// TIA Portal project "babu_counterBasics" (V15)

(* hardware
DEVICE "S7-1200 station_1"  S7-1200 Station
   slot 0: "Rack_0"  S7-1200 Rack  Rack  V1.0
   slot 1: "PLC_1"  CPU 1212C DC/DC/DC  6ES7 212-1AE40-0XB0  V4.2
*)

// ===== PLC "PLC_1"  CPU 1212C DC/DC/DC =====

VAR_GLOBAL   // PLC tag table "Default tag table"
   "sensor" AT %M0.0 : Bool;
   "reset" AT %M0.1 : Bool;
   "Tag_3" AT %MW0 : Int;
   "indicator light" AT %Q0.0 : Bool;
   "load" AT %M0.2 : Bool;
   "START PULSE 2" AT %M2.0 : Bool;
   "PULSE OUTPUT 2" AT %M2.1 : Bool;
   "START MEMORY" AT %M2.2 : Bool;
   "START MEMORY 2" AT %M2.3 : Bool;
   "TIMER MEMORY" AT %M2.4 : Bool;
   "COUNTER UP OUTPUT" AT %Q0.1 : Bool;
   "RESET CU" AT %M2.5 : Bool;
   "COUNTER DOWN OUTPUT" AT %Q0.2 : Bool;
   "LOAD DATA COUNTER DOWN" AT %M2.6 : Bool;
   "INITIALIZE" AT %M2.7 : Bool;
   "COUNTER UP DOWN OUTPUT" AT %M3.0 : Bool;
   "COUNTER DOWN RESET 5" AT %M3.1 : Bool;
   "COUNTER DOWN LOAD 5" AT %M3.2 : Bool;
   "COUNTER UP DOWN RESET" AT %M3.3 : Bool;
   "COUNTER DOWN 5" AT %M3.4 : Bool;
   "COUNTER DOWN OUTPUT 5" AT %M3.5 : Bool;
   "COUNTER DOWN SET 5" AT %M3.6 : Bool;
   "START 6" AT %M3.7 : Bool;
   "UP DOWN LONG PULSE" AT %M4.0 : Bool;
   "UP DOWN LONG PULSE MEM" AT %M4.1 : Bool;
   "COUNT UP" AT %M4.2 : Bool;
   "COUNT DOWN" AT %M4.3 : Bool;
   "COUNT DOWN TEMP" AT %M4.4 : Bool;
   "COUNTER UP OUTPUT 5" AT %M4.5 : Bool;
END_VAR

// folder: System blocks/Program resources

DATA_BLOCK "IEC_Counter_0_DB"   // DB1
{ S7_Optimized_Access := 'TRUE' }
AUTHOR : Simatic
FAMILY : IEC
NAME : CNTR
VERSION : 1.0
// stored: InstanceOfName IEC_COUNTER
"IEC_COUNTER"
BEGIN
END_DATA_BLOCK

DATA_BLOCK "IEC_Timer_0_DB_2"   // DB2
{ S7_Optimized_Access := 'TRUE' }
AUTHOR : Simatic
FAMILY : IEC
NAME : IEC_TMR
VERSION : 1.0
// stored: InstanceOfName IEC_TIMER
"IEC_TIMER"
BEGIN
END_DATA_BLOCK

DATA_BLOCK "IEC_Timer_0_DB"   // DB3
{ S7_Optimized_Access := 'TRUE' }
AUTHOR : Simatic
FAMILY : IEC
NAME : IEC_TMR
VERSION : 1.0
// stored: InstanceOfName IEC_TIMER
"IEC_TIMER"
BEGIN
END_DATA_BLOCK

DATA_BLOCK "IEC_Timer_0_DB_1"   // DB4
{ S7_Optimized_Access := 'TRUE' }
AUTHOR : Simatic
FAMILY : IEC
NAME : IEC_TMR
VERSION : 1.0
// stored: InstanceOfName IEC_TIMER
"IEC_TIMER"
BEGIN
END_DATA_BLOCK

DATA_BLOCK "IEC_Counter_0_DB_1"   // DB5
{ S7_Optimized_Access := 'TRUE' }
AUTHOR : Simatic
FAMILY : IEC
NAME : CNTR
VERSION : 1.0
// stored: InstanceOfName IEC_COUNTER
"IEC_COUNTER"
BEGIN
END_DATA_BLOCK

DATA_BLOCK "IEC_Timer_0_DB_3"   // DB6
{ S7_Optimized_Access := 'TRUE' }
AUTHOR : Simatic
FAMILY : IEC
NAME : IEC_TMR
VERSION : 1.0
// stored: InstanceOfName IEC_TIMER
"IEC_TIMER"
BEGIN
END_DATA_BLOCK

DATA_BLOCK "IEC_Counter_0_DB_2"   // DB7
{ S7_Optimized_Access := 'TRUE' }
AUTHOR : Simatic
FAMILY : IEC
NAME : CNTR
VERSION : 1.0
// stored: InstanceOfName IEC_COUNTER
"IEC_COUNTER"
BEGIN
END_DATA_BLOCK

DATA_BLOCK "IEC_Timer_0_DB_4"   // DB8
{ S7_Optimized_Access := 'TRUE' }
AUTHOR : Simatic
FAMILY : IEC
NAME : IEC_TMR
VERSION : 1.0
// stored: InstanceOfName IEC_TIMER
"IEC_TIMER"
BEGIN
END_DATA_BLOCK

DATA_BLOCK "IEC_Timer_0_DB_5"   // DB9
{ S7_Optimized_Access := 'TRUE' }
AUTHOR : Simatic
FAMILY : IEC
NAME : IEC_TMR
VERSION : 1.0
// stored: InstanceOfName IEC_TIMER
"IEC_TIMER"
BEGIN
END_DATA_BLOCK

DATA_BLOCK "IEC_Counter_0_DB_3"   // DB10
{ S7_Optimized_Access := 'TRUE' }
AUTHOR : Simatic
FAMILY : IEC
NAME : CNTR
VERSION : 1.0
// stored: InstanceOfName IEC_COUNTER
"IEC_COUNTER"
BEGIN
END_DATA_BLOCK

DATA_BLOCK "IEC_Timer_0_DB_6"   // DB11
{ S7_Optimized_Access := 'TRUE' }
AUTHOR : Simatic
FAMILY : IEC
NAME : IEC_TMR
VERSION : 1.0
// stored: InstanceOfName IEC_TIMER
"IEC_TIMER"
BEGIN
END_DATA_BLOCK

DATA_BLOCK "IEC_Timer_0_DB_8"   // DB13
{ S7_Optimized_Access := 'TRUE' }
AUTHOR : Simatic
FAMILY : IEC
NAME : IEC_TMR
VERSION : 1.0
// stored: InstanceOfName IEC_TIMER
"IEC_TIMER"
BEGIN
END_DATA_BLOCK

DATA_BLOCK "IEC_Timer_0_DB_9"   // DB14
{ S7_Optimized_Access := 'TRUE' }
AUTHOR : Simatic
FAMILY : IEC
NAME : IEC_TMR
VERSION : 1.0
// stored: InstanceOfName IEC_TIMER
"IEC_TIMER"
BEGIN
END_DATA_BLOCK

DATA_BLOCK "IEC_Timer_0_DB_10"   // DB15
{ S7_Optimized_Access := 'TRUE' }
AUTHOR : Simatic
FAMILY : IEC
NAME : IEC_TMR
VERSION : 1.0
// stored: InstanceOfName IEC_TIMER
"IEC_TIMER"
BEGIN
END_DATA_BLOCK

DATA_BLOCK "IEC_Timer_0_DB_12"   // DB17
{ S7_Optimized_Access := 'TRUE' }
AUTHOR : Simatic
FAMILY : IEC
NAME : IEC_TMR
VERSION : 1.0
// stored: InstanceOfName IEC_TIMER
"IEC_TIMER"
BEGIN
END_DATA_BLOCK

DATA_BLOCK "IEC_Timer_0_DB_13"   // DB18
{ S7_Optimized_Access := 'TRUE' }
AUTHOR : Simatic
FAMILY : IEC
NAME : IEC_TMR
VERSION : 1.0
// stored: InstanceOfName IEC_TIMER
"IEC_TIMER"
BEGIN
END_DATA_BLOCK

DATA_BLOCK "IEC_Timer_0_DB_14"   // DB19
{ S7_Optimized_Access := 'TRUE' }
AUTHOR : Simatic
FAMILY : IEC
NAME : IEC_TMR
VERSION : 1.0
// stored: InstanceOfName IEC_TIMER
"IEC_TIMER"
BEGIN
END_DATA_BLOCK

DATA_BLOCK "IEC_Timer_0_DB_15"   // DB20
{ S7_Optimized_Access := 'TRUE' }
AUTHOR : Simatic
FAMILY : IEC
NAME : IEC_TMR
VERSION : 1.0
// stored: InstanceOfName IEC_TIMER
"IEC_TIMER"
BEGIN
END_DATA_BLOCK

// folder: (top level)

ORGANIZATION_BLOCK "Main"   // OB1, LAD, ProgramCycle
TITLE = "Main Program Sweep (Cycle)"
{ S7_Optimized_Access := 'TRUE' }
VERSION : 0.1
   VAR_INPUT
      Initial_Call : Bool;   // Initial call of this OB
      Remanence : Bool;   // =True, if remanent data are available
   END_VAR
   VAR_TEMP   // added for the SCL form of the ladder/FBD networks
      _w1 : Bool;
      _w2 : Bool;
   END_VAR
BEGIN

REGION Network 1
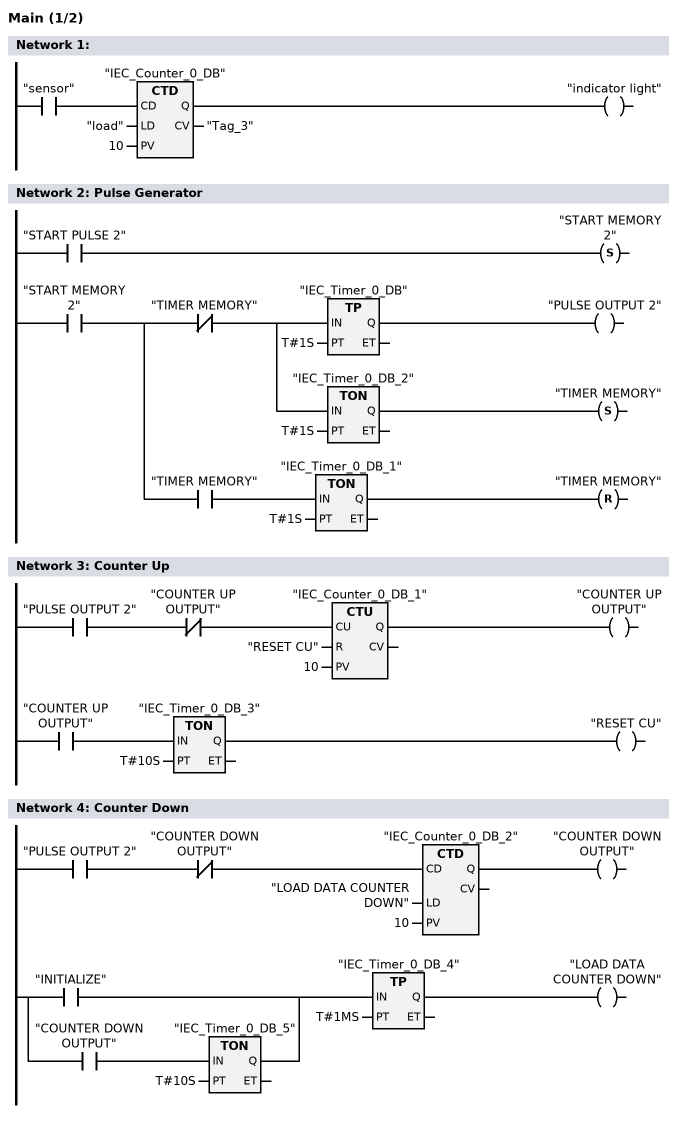
   "IEC_Counter_0_DB".CTD(CD := "sensor", LD := "load", PV := 10, CV => "Tag_3");
   "indicator light" := "IEC_Counter_0_DB".Q;
END_REGION

REGION Network 2: Pulse Generator
   IF "START PULSE 2" THEN "START MEMORY 2" := TRUE; END_IF;
   #_w1 := "START MEMORY 2" AND NOT "TIMER MEMORY";
   "IEC_Timer_0_DB".TP(IN := #_w1, PT := T#1S);
   "PULSE OUTPUT 2" := "IEC_Timer_0_DB".Q;
   "IEC_Timer_0_DB_2".TON(IN := #_w1, PT := T#1S);
   IF "IEC_Timer_0_DB_2".Q THEN "TIMER MEMORY" := TRUE; END_IF;
   "IEC_Timer_0_DB_1".TON(IN := "START MEMORY 2" AND "TIMER MEMORY", PT := T#1S);
   IF "IEC_Timer_0_DB_1".Q THEN "TIMER MEMORY" := FALSE; END_IF;
END_REGION

REGION Network 3: Counter Up
   "IEC_Counter_0_DB_1".CTU(CU := "PULSE OUTPUT 2" AND NOT "COUNTER UP OUTPUT", R := "RESET CU", PV := 10);
   "COUNTER UP OUTPUT" := "IEC_Counter_0_DB_1".Q;
   "IEC_Timer_0_DB_3".TON(IN := "COUNTER UP OUTPUT", PT := T#10S);
   "RESET CU" := "IEC_Timer_0_DB_3".Q;
END_REGION

REGION Network 4: Counter Down
   "IEC_Counter_0_DB_2".CTD(CD := "PULSE OUTPUT 2" AND NOT "COUNTER DOWN OUTPUT",
                           LD := "LOAD DATA COUNTER DOWN",
                           PV := 10);
   "COUNTER DOWN OUTPUT" := "IEC_Counter_0_DB_2".Q;
   "IEC_Timer_0_DB_5".TON(IN := "COUNTER DOWN OUTPUT", PT := T#10S);
   "IEC_Timer_0_DB_4".TP(IN := "INITIALIZE" OR "IEC_Timer_0_DB_5".Q, PT := T#1MS);
   "LOAD DATA COUNTER DOWN" := "IEC_Timer_0_DB_4".Q;
END_REGION

REGION Network 5: COUNTER UP DOWN
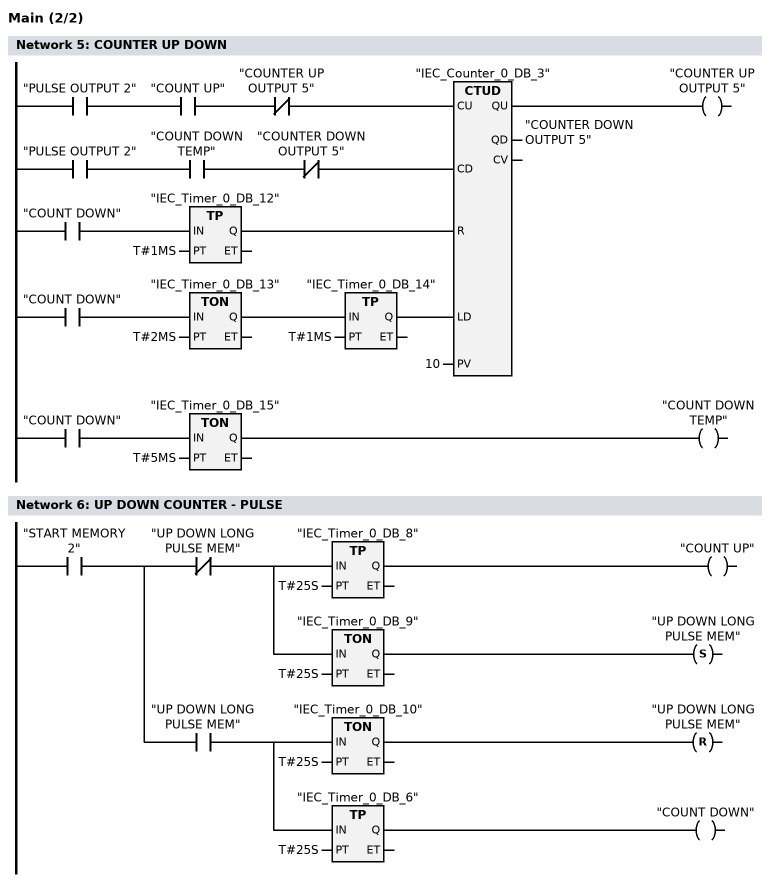
   "IEC_Timer_0_DB_12".TP(IN := "COUNT DOWN", PT := T#1MS);
   "IEC_Timer_0_DB_13".TON(IN := "COUNT DOWN", PT := T#2MS);
   "IEC_Timer_0_DB_14".TP(IN := "IEC_Timer_0_DB_13".Q, PT := T#1MS);
   "IEC_Counter_0_DB_3".CTUD(CU := "PULSE OUTPUT 2" AND "COUNT UP" AND NOT "COUNTER UP OUTPUT 5",
                           CD := "PULSE OUTPUT 2" AND "COUNT DOWN TEMP" AND NOT "COUNTER DOWN OUTPUT 5",
                           R := "IEC_Timer_0_DB_12".Q,
                           LD := "IEC_Timer_0_DB_14".Q,
                           PV := 10,
                           QD => "COUNTER DOWN OUTPUT 5");
   "COUNTER UP OUTPUT 5" := "IEC_Counter_0_DB_3".QU;
   "IEC_Timer_0_DB_15".TON(IN := "COUNT DOWN", PT := T#5MS);
   "COUNT DOWN TEMP" := "IEC_Timer_0_DB_15".Q;
END_REGION

REGION Network 6: UP DOWN COUNTER - PULSE
   #_w1 := "START MEMORY 2" AND NOT "UP DOWN LONG PULSE MEM";
   "IEC_Timer_0_DB_8".TP(IN := #_w1, PT := T#25S);
   "COUNT UP" := "IEC_Timer_0_DB_8".Q;
   "IEC_Timer_0_DB_9".TON(IN := #_w1, PT := T#25S);
   IF "IEC_Timer_0_DB_9".Q THEN "UP DOWN LONG PULSE MEM" := TRUE; END_IF;
   #_w2 := "START MEMORY 2" AND "UP DOWN LONG PULSE MEM";
   "IEC_Timer_0_DB_10".TON(IN := #_w2, PT := T#25S);
   IF "IEC_Timer_0_DB_10".Q THEN "UP DOWN LONG PULSE MEM" := FALSE; END_IF;
   "IEC_Timer_0_DB_6".TP(IN := #_w2, PT := T#25S);
   "COUNT DOWN" := "IEC_Timer_0_DB_6".Q;
END_REGION
END_ORGANIZATION_BLOCK